Staubli VAL3: math.pjx

--- math.pjx ---
Parameters version=s8.13.1Cs9_BS2800 stackSize=5000 millimeterUnit=true
Program file=cumsum.pgx
Program file=diff.pgx
Program file=rollsum.pgx
Program file=root.pgx
Program file=sign.pgx
Program file=square.pgx
Program file=start.pgx
Program file=stop.pgx
Program file=sum.pgx
Data file=math.dtx
Library alias=utils path=Disk://helpers/helpers.pjx

--- math.dtx ---
num nResult
num nIndex
num nResult2
num nTest[7]
num nResultTest

--- start.pgx ---
program start()
begin

  nTest[0] = 0
  nTest[1] = 2
  nTest[2] = -4
  nTest[3] = 10
  nTest[5] = -3
  nTest[6] = 4

  call rollsum(nTest, 3,nResultTest)

end

--- cumsum.pgx ---
public program cumsum(num& x_nInput[], num& x_nResult[])
  local num l_nLength
  local num l_nElement
begin

  l_nLength = size(x_nInput)
  x_nResult[0] = 0
  resize(x_nResult,1,l_nLength)

  for l_nElement = 0 to l_nLength-1
    if l_nElement == 0
      x_nResult[0] = x_nInput[0]
    else
      x_nResult[l_nElement] = x_nResult[l_nElement-1] + x_nInput[l_nElement]
    endIf

  endFor

end

--- diff.pgx ---
public program diff(num& x_nInput[], num& x_nResult[])
  local num l_nLength
  local num l_nElement
begin

  l_nLength = size(x_nInput)
  x_nResult[0] = 0
  resize(x_nResult,1,l_nLength-1)

  for l_nElement = 1 to l_nLength-1
    x_nResult[l_nElement-1] =  x_nInput[l_nElement] - x_nInput[l_nElement-1]
  endFor

end

--- rollsum.pgx ---
public program rollsum(num& x_nInput[], num x_nWindow, num& x_nResult[])
  local num l_nLength
  local num l_nElement
  local num l_nSum
begin

  l_nLength = size(x_nInput)
  x_nResult = 0
  resize(x_nResult,1,l_nLength-x_nWindow+1)

  l_nElement = 0
  while l_nElement <l_nLength-x_nWindow+1
    call utils:range(l_nElement, l_nElement+x_nWindow, 1,nIndex)
    call utils:extractNum(x_nInput,nIndex,nResult)
    call sum(nResult, l_nSum)

    x_nResult[l_nElement] = l_nSum
    l_nElement = l_nElement + 1
  endWhile

end

--- root.pgx ---
public program root(num& x_nInput[], num& x_nResult[])
  local num l_nLength
  local num l_nElement
begin

  l_nLength = size(x_nInput)
  resize(x_nResult,1,1)
  x_nResult = 0
  resize(x_nResult,1,l_nLength)

  for l_nElement = 0 to l_nLength -1
    x_nResult[l_nElement] = power(x_nInput[l_nElement],0.5)
  endFor

end

--- sign.pgx ---
public program sign()
begin
end

--- square.pgx ---
public program square(num& x_nInput[], num& x_nResult[])
  local num l_nLength
  local num l_nElement
begin

  l_nLength = size(x_nInput)
  resize(x_nResult,1,1)
  x_nResult = 0
  resize(x_nResult,1,l_nLength)

  for l_nElement = 0 to l_nLength -1
    x_nResult[l_nElement] = x_nInput[l_nElement]*x_nInput[l_nElement]
  endFor

end

--- sum.pgx ---
public program sum(num& x_nInput[], num& x_nResult)
  local num l_nLength
  local num l_nElement
begin

  l_nLength = size(x_nInput)
  x_nResult = 0

  for l_nElement = 0 to l_nLength-1
    x_nResult = x_nResult + x_nInput[l_nElement]
  endFor

end
